// Mitsubishi GX Works2 project: test   PLC: Q00

// global labels: Global1
VAR_GLOBAL
  Start AT M1 : BOOL;
  Motor AT Y0 : BOOL;
  MV_Turtall AT D1 : INT;
  SP_Turtall AT D0 : INT;
  Stopp AT M0 : BOOL;
END_VAR

// task Task_01 (event TRUE, interval 0, priority 31): POU_01

PROGRAM POU_01
(* structured ladder/FBD written out as ST: instructions are called as NAME(EN, inputs, outputs); _pN, _eN, _tN stand for wires *)
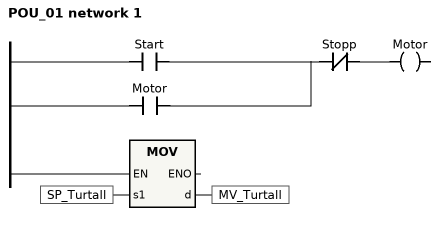
(* network 1 *)
Motor := (Start OR Motor) AND NOT Stopp;
MOV(TRUE, SP_Turtall, MV_Turtall);
END_PROGRAM
